Staubli VAL3: SoapTestScan.dtx

bool bSignal
bool bTxt1
bool bTxt2
bool bTxt3
bool btrig
public dio fout = {link=fOut0}
public frame FrmDraw = {x=1000, y=-50, fatherId=world[0]}
mdesc mNomSpeed
num l_nInit = 1500
public num nByteOut[48]
num nNumTotal = 5031
num nNumrecord = 5031
public num nTranC[6]
  [0] = -21.496
  [1] = -9.92
  [2] = 104.826
  [3] = 179.902
  [4] = 0.184
  [5] = -123.901
num nTxtTotal = 11
num n_sTxt = 1
num ndelay = 91.328
public num nnnn
num ntime = 653.375
public pointRx shere = {x=-21.496, y=-9.92, z=104.826, rx=179.902, ry=0.184, rz=-123.901, fatherId=FrmDraw[0]}
public sio sSocketout = {link=Socket\CServerSocket}
tool tTool = {fatherId=flange[0], ioLink=valve1}
public num hpn
public num lpn
public num ppn
num very
public num hery
public num pery
public num zmin
public num ymin
public num xmin
public num zmax
public num ymax
public num xmax
public num ztp
public num ytp
public num xtp
public num xore
public num yore
public num zore
public num nMenu
public num Qery
string sTap[3000]
string sString[1500]
public pointRx pfrmCad[1500]
  [0] = {fatherId=world[0]}
  [1] = {fatherId=world[0]}
  [2] = {fatherId=world[0]}
  [3] = {fatherId=world[0]}
  [4] = {fatherId=world[0]}
  [5] = {fatherId=world[0]}
  [6] = {fatherId=world[0]}
  [7] = {fatherId=world[0]}
  [8] = {fatherId=world[0]}
  [9] = {fatherId=world[0]}
  [10] = {fatherId=world[0]}
  [11] = {fatherId=world[0]}
  [12] = {fatherId=world[0]}
  [13] = {fatherId=world[0]}
  [14] = {fatherId=world[0]}
  [15] = {fatherId=world[0]}
  [16] = {fatherId=world[0]}
  [17] = {fatherId=world[0]}
  [18] = {fatherId=world[0]}
  [19] = {fatherId=world[0]}
  [20] = {fatherId=world[0]}
  [21] = {fatherId=world[0]}
  [22] = {fatherId=world[0]}
  [23] = {fatherId=world[0]}
  [24] = {fatherId=world[0]}
  [25] = {fatherId=world[0]}
  [26] = {fatherId=world[0]}
  [27] = {fatherId=world[0]}
  [28] = {fatherId=world[0]}
  [29] = {fatherId=world[0]}
  [30] = {fatherId=world[0]}
  [31] = {fatherId=world[0]}
  [32] = {fatherId=world[0]}
  [33] = {fatherId=world[0]}
  [34] = {fatherId=world[0]}
  [35] = {fatherId=world[0]}
  [36] = {fatherId=world[0]}
  [37] = {fatherId=world[0]}
  [38] = {fatherId=world[0]}
  [39] = {fatherId=world[0]}
  [40] = {fatherId=world[0]}
  [41] = {fatherId=world[0]}
  [42] = {fatherId=world[0]}
  [43] = {fatherId=world[0]}
  [44] = {fatherId=world[0]}
  [45] = {fatherId=world[0]}
  [46] = {fatherId=world[0]}
  [47] = {fatherId=world[0]}
  [48] = {fatherId=world[0]}
  [49] = {fatherId=world[0]}
  [50] = {fatherId=world[0]}
  [51] = {fatherId=world[0]}
  [52] = {fatherId=world[0]}
  [53] = {fatherId=world[0]}
  [54] = {fatherId=world[0]}
  [55] = {fatherId=world[0]}
  [56] = {fatherId=world[0]}
  [57] = {fatherId=world[0]}
  [58] = {fatherId=world[0]}
  [59] = {fatherId=world[0]}
  [60] = {fatherId=world[0]}
  [61] = {fatherId=world[0]}
  [62] = {fatherId=world[0]}
  [63] = {fatherId=world[0]}
  [64] = {fatherId=world[0]}
  [65] = {fatherId=world[0]}
  [66] = {fatherId=world[0]}
  [67] = {fatherId=world[0]}
  [68] = {fatherId=world[0]}
  [69] = {fatherId=world[0]}
  [70] = {fatherId=world[0]}
  [71] = {fatherId=world[0]}
  [72] = {fatherId=world[0]}
  [73] = {fatherId=world[0]}
  [74] = {fatherId=world[0]}
  [75] = {fatherId=world[0]}
  [76] = {fatherId=world[0]}
  [77] = {fatherId=world[0]}
  [78] = {fatherId=world[0]}
  [79] = {fatherId=world[0]}
  [80] = {fatherId=world[0]}
  [81] = {fatherId=world[0]}
  [82] = {fatherId=world[0]}
  [83] = {fatherId=world[0]}
  [84] = {fatherId=world[0]}
  [85] = {fatherId=world[0]}
  [86] = {fatherId=world[0]}
  [87] = {fatherId=world[0]}
  [88] = {fatherId=world[0]}
  [89] = {fatherId=world[0]}
  [90] = {fatherId=world[0]}
  [91] = {fatherId=world[0]}
  [92] = {fatherId=world[0]}
  [93] = {fatherId=world[0]}
  [94] = {fatherId=world[0]}
  [95] = {fatherId=world[0]}
  [96] = {fatherId=world[0]}
  [97] = {fatherId=world[0]}
  [98] = {fatherId=world[0]}
  [99] = {fatherId=world[0]}
  [100] = {fatherId=world[0]}
  [101] = {fatherId=world[0]}
  [102] = {fatherId=world[0]}
  [103] = {fatherId=world[0]}
  [104] = {fatherId=world[0]}
  [105] = {fatherId=world[0]}
  [106] = {fatherId=world[0]}
  [107] = {fatherId=world[0]}
  [108] = {fatherId=world[0]}
  [109] = {fatherId=world[0]}
  [110] = {fatherId=world[0]}
  [111] = {fatherId=world[0]}
  [112] = {fatherId=world[0]}
  [113] = {fatherId=world[0]}
  [114] = {fatherId=world[0]}
  [115] = {fatherId=world[0]}
  [116] = {fatherId=world[0]}
  [117] = {fatherId=world[0]}
  [118] = {fatherId=world[0]}
  [119] = {fatherId=world[0]}
  [120] = {fatherId=world[0]}
  [121] = {fatherId=world[0]}
  [122] = {fatherId=world[0]}
  [123] = {fatherId=world[0]}
  [124] = {fatherId=world[0]}
  [125] = {fatherId=world[0]}
  [126] = {fatherId=world[0]}
  [127] = {fatherId=world[0]}
  [128] = {fatherId=world[0]}
  [129] = {fatherId=world[0]}
  [130] = {fatherId=world[0]}
  [131] = {fatherId=world[0]}
  [132] = {fatherId=world[0]}
  [133] = {fatherId=world[0]}
  [134] = {fatherId=world[0]}
  [135] = {fatherId=world[0]}
  [136] = {fatherId=world[0]}
  [137] = {fatherId=world[0]}
  [138] = {fatherId=world[0]}
  [139] = {fatherId=world[0]}
  [140] = {fatherId=world[0]}
  [141] = {fatherId=world[0]}
  [142] = {fatherId=world[0]}
  [143] = {fatherId=world[0]}
  [144] = {fatherId=world[0]}
  [145] = {fatherId=world[0]}
  [146] = {fatherId=world[0]}
  [147] = {fatherId=world[0]}
  [148] = {fatherId=world[0]}
  [149] = {fatherId=world[0]}
  [150] = {fatherId=world[0]}
  [151] = {fatherId=world[0]}
  [152] = {fatherId=world[0]}
  [153] = {fatherId=world[0]}
  [154] = {fatherId=world[0]}
  [155] = {fatherId=world[0]}
  [156] = {fatherId=world[0]}
  [157] = {fatherId=world[0]}
  [158] = {fatherId=world[0]}
  [159] = {fatherId=world[0]}
  [160] = {fatherId=world[0]}
  [161] = {fatherId=world[0]}
  [162] = {fatherId=world[0]}
  [163] = {fatherId=world[0]}
  [164] = {fatherId=world[0]}
  [165] = {fatherId=world[0]}
  [166] = {fatherId=world[0]}
  [167] = {fatherId=world[0]}
  [168] = {fatherId=world[0]}
  [169] = {fatherId=world[0]}
  [170] = {fatherId=world[0]}
  [171] = {fatherId=world[0]}
  [172] = {fatherId=world[0]}
  [173] = {fatherId=world[0]}
  [174] = {fatherId=world[0]}
  [175] = {fatherId=world[0]}
  [176] = {fatherId=world[0]}
  [177] = {fatherId=world[0]}
  [178] = {fatherId=world[0]}
  [179] = {fatherId=world[0]}
  [180] = {fatherId=world[0]}
  [181] = {fatherId=world[0]}
  [182] = {fatherId=world[0]}
  [183] = {fatherId=world[0]}
  [184] = {fatherId=world[0]}
  [185] = {fatherId=world[0]}
  [186] = {fatherId=world[0]}
  [187] = {fatherId=world[0]}
  [188] = {fatherId=world[0]}
  [189] = {fatherId=world[0]}
  [190] = {fatherId=world[0]}
  [191] = {fatherId=world[0]}
  [192] = {fatherId=world[0]}
  [193] = {fatherId=world[0]}
  [194] = {fatherId=world[0]}
  [195] = {fatherId=world[0]}
  [196] = {fatherId=world[0]}
  [197] = {fatherId=world[0]}
  [198] = {fatherId=world[0]}
  [199] = {fatherId=world[0]}
  [200] = {fatherId=world[0]}
  [201] = {fatherId=world[0]}
  [202] = {fatherId=world[0]}
  [203] = {fatherId=world[0]}
  [204] = {fatherId=world[0]}
  [205] = {fatherId=world[0]}
  [206] = {fatherId=world[0]}
  [207] = {fatherId=world[0]}
  [208] = {fatherId=world[0]}
  [209] = {fatherId=world[0]}
  [210] = {fatherId=world[0]}
  [211] = {fatherId=world[0]}
  [212] = {fatherId=world[0]}
  [213] = {fatherId=world[0]}
  [214] = {fatherId=world[0]}
  [215] = {fatherId=world[0]}
  [216] = {fatherId=world[0]}
  [217] = {fatherId=world[0]}
  [218] = {fatherId=world[0]}
  [219] = {fatherId=world[0]}
  [220] = {fatherId=world[0]}
  [221] = {fatherId=world[0]}
  [222] = {fatherId=world[0]}
  [223] = {fatherId=world[0]}
  [224] = {fatherId=world[0]}
  [225] = {fatherId=world[0]}
  [226] = {fatherId=world[0]}
  [227] = {fatherId=world[0]}
  [228] = {fatherId=world[0]}
  [229] = {fatherId=world[0]}
  [230] = {fatherId=world[0]}
  [231] = {fatherId=world[0]}
  [232] = {fatherId=world[0]}
  [233] = {fatherId=world[0]}
  [234] = {fatherId=world[0]}
  [235] = {fatherId=world[0]}
  [236] = {fatherId=world[0]}
  [237] = {fatherId=world[0]}
  [238] = {fatherId=world[0]}
  [239] = {fatherId=world[0]}
  [240] = {fatherId=world[0]}
  [241] = {fatherId=world[0]}
  [242] = {fatherId=world[0]}
  [243] = {fatherId=world[0]}
  [244] = {fatherId=world[0]}
  [245] = {fatherId=world[0]}
  [246] = {fatherId=world[0]}
  [247] = {fatherId=world[0]}
  [248] = {fatherId=world[0]}
  [249] = {fatherId=world[0]}
  [250] = {fatherId=world[0]}
  [251] = {fatherId=world[0]}
  [252] = {fatherId=world[0]}
  [253] = {fatherId=world[0]}
  [254] = {fatherId=world[0]}
  [255] = {fatherId=world[0]}
  [256] = {fatherId=world[0]}
  [257] = {fatherId=world[0]}
  [258] = {fatherId=world[0]}
  [259] = {fatherId=world[0]}
  [260] = {fatherId=world[0]}
  [261] = {fatherId=world[0]}
  [262] = {fatherId=world[0]}
  [263] = {fatherId=world[0]}
  [264] = {fatherId=world[0]}
  [265] = {fatherId=world[0]}
  [266] = {fatherId=world[0]}
  [267] = {fatherId=world[0]}
  [268] = {fatherId=world[0]}
  [269] = {fatherId=world[0]}
  [270] = {fatherId=world[0]}
  [271] = {fatherId=world[0]}
  [272] = {fatherId=world[0]}
  [273] = {fatherId=world[0]}
  [274] = {fatherId=world[0]}
  [275] = {fatherId=world[0]}
  [276] = {fatherId=world[0]}
  [277] = {fatherId=world[0]}
  [278] = {fatherId=world[0]}
  [279] = {fatherId=world[0]}
  [280] = {fatherId=world[0]}
  [281] = {fatherId=world[0]}
  [282] = {fatherId=world[0]}
  [283] = {fatherId=world[0]}
  [284] = {fatherId=world[0]}
  [285] = {fatherId=world[0]}
  [286] = {fatherId=world[0]}
  [287] = {fatherId=world[0]}
  [288] = {fatherId=world[0]}
  [289] = {fatherId=world[0]}
  [290] = {fatherId=world[0]}
  [291] = {fatherId=world[0]}
  [292] = {fatherId=world[0]}
  [293] = {fatherId=world[0]}
  [294] = {fatherId=world[0]}
  [295] = {fatherId=world[0]}
  [296] = {fatherId=world[0]}
  [297] = {fatherId=world[0]}
  [298] = {fatherId=world[0]}
  [299] = {fatherId=world[0]}
  [300] = {fatherId=world[0]}
  [301] = {fatherId=world[0]}
  [302] = {fatherId=world[0]}
  [303] = {fatherId=world[0]}
  [304] = {fatherId=world[0]}
  [305] = {fatherId=world[0]}
  [306] = {fatherId=world[0]}
  [307] = {fatherId=world[0]}
  [308] = {fatherId=world[0]}
  [309] = {fatherId=world[0]}
  [310] = {fatherId=world[0]}
  [311] = {fatherId=world[0]}
  [312] = {fatherId=world[0]}
  [313] = {fatherId=world[0]}
  [314] = {fatherId=world[0]}
  [315] = {fatherId=world[0]}
  [316] = {fatherId=world[0]}
  [317] = {fatherId=world[0]}
  [318] = {fatherId=world[0]}
  [319] = {fatherId=world[0]}
  [320] = {fatherId=world[0]}
  [321] = {fatherId=world[0]}
  [322] = {fatherId=world[0]}
  [323] = {fatherId=world[0]}
  [324] = {fatherId=world[0]}
  [325] = {fatherId=world[0]}
  [326] = {fatherId=world[0]}
  [327] = {fatherId=world[0]}
  [328] = {fatherId=world[0]}
  [329] = {fatherId=world[0]}
  [330] = {fatherId=world[0]}
  [331] = {fatherId=world[0]}
  [332] = {fatherId=world[0]}
  [333] = {fatherId=world[0]}
  [334] = {fatherId=world[0]}
  [335] = {fatherId=world[0]}
  [336] = {fatherId=world[0]}
  [337] = {fatherId=world[0]}
  [338] = {fatherId=world[0]}
  [339] = {fatherId=world[0]}
  [340] = {fatherId=world[0]}
  [341] = {fatherId=world[0]}
  [342] = {fatherId=world[0]}
  [343] = {fatherId=world[0]}
  [344] = {fatherId=world[0]}
  [345] = {fatherId=world[0]}
  [346] = {fatherId=world[0]}
  [347] = {fatherId=world[0]}
  [348] = {fatherId=world[0]}
  [349] = {fatherId=world[0]}
  [350] = {fatherId=world[0]}
  [351] = {fatherId=world[0]}
  [352] = {fatherId=world[0]}
  [353] = {fatherId=world[0]}
  [354] = {fatherId=world[0]}
  [355] = {fatherId=world[0]}
  [356] = {fatherId=world[0]}
  [357] = {fatherId=world[0]}
  [358] = {fatherId=world[0]}
  [359] = {fatherId=world[0]}
  [360] = {fatherId=world[0]}
  [361] = {fatherId=world[0]}
  [362] = {fatherId=world[0]}
  [363] = {fatherId=world[0]}
  [364] = {fatherId=world[0]}
  [365] = {fatherId=world[0]}
  [366] = {fatherId=world[0]}
  [367] = {fatherId=world[0]}
  [368] = {fatherId=world[0]}
  [369] = {fatherId=world[0]}
  [370] = {fatherId=world[0]}
  [371] = {fatherId=world[0]}
  [372] = {fatherId=world[0]}
  [373] = {fatherId=world[0]}
  [374] = {fatherId=world[0]}
  [375] = {fatherId=world[0]}
  [376] = {fatherId=world[0]}
  [377] = {fatherId=world[0]}
  [378] = {fatherId=world[0]}
  [379] = {fatherId=world[0]}
  [380] = {fatherId=world[0]}
  [381] = {fatherId=world[0]}
  [382] = {fatherId=world[0]}
  [383] = {fatherId=world[0]}
  [384] = {fatherId=world[0]}
  [385] = {fatherId=world[0]}
  [386] = {fatherId=world[0]}
  [387] = {fatherId=world[0]}
  [388] = {fatherId=world[0]}
  [389] = {fatherId=world[0]}
  [390] = {fatherId=world[0]}
  [391] = {fatherId=world[0]}
  [392] = {fatherId=world[0]}
  [393] = {fatherId=world[0]}
  [394] = {fatherId=world[0]}
  [395] = {fatherId=world[0]}
  [396] = {fatherId=world[0]}
  [397] = {fatherId=world[0]}
  [398] = {fatherId=world[0]}
  [399] = {fatherId=world[0]}
  [400] = {fatherId=world[0]}
  [401] = {fatherId=world[0]}
  [402] = {fatherId=world[0]}
  [403] = {fatherId=world[0]}
  [404] = {fatherId=world[0]}
  [405] = {fatherId=world[0]}
  [406] = {fatherId=world[0]}
  [407] = {fatherId=world[0]}
  [408] = {fatherId=world[0]}
  [409] = {fatherId=world[0]}
  [410] = {fatherId=world[0]}
  [411] = {fatherId=world[0]}
  [412] = {fatherId=world[0]}
  [413] = {fatherId=world[0]}
  [414] = {fatherId=world[0]}
  [415] = {fatherId=world[0]}
  [416] = {fatherId=world[0]}
  [417] = {fatherId=world[0]}
  [418] = {fatherId=world[0]}
  [419] = {fatherId=world[0]}
  [420] = {fatherId=world[0]}
  [421] = {fatherId=world[0]}
  [422] = {fatherId=world[0]}
  [423] = {fatherId=world[0]}
  [424] = {fatherId=world[0]}
  [425] = {fatherId=world[0]}
  [426] = {fatherId=world[0]}
  [427] = {fatherId=world[0]}
  [428] = {fatherId=world[0]}
  [429] = {fatherId=world[0]}
  [430] = {fatherId=world[0]}
  [431] = {fatherId=world[0]}
  [432] = {fatherId=world[0]}
  [433] = {fatherId=world[0]}
  [434] = {fatherId=world[0]}
  [435] = {fatherId=world[0]}
  [436] = {fatherId=world[0]}
  [437] = {fatherId=world[0]}
  [438] = {fatherId=world[0]}
  [439] = {fatherId=world[0]}
  [440] = {fatherId=world[0]}
  [441] = {fatherId=world[0]}
  [442] = {fatherId=world[0]}
  [443] = {fatherId=world[0]}
  [444] = {fatherId=world[0]}
  [445] = {fatherId=world[0]}
  [446] = {fatherId=world[0]}
  [447] = {fatherId=world[0]}
  [448] = {fatherId=world[0]}
  [449] = {fatherId=world[0]}
  [450] = {fatherId=world[0]}
  [451] = {fatherId=world[0]}
  [452] = {fatherId=world[0]}
  [453] = {fatherId=world[0]}
  [454] = {fatherId=world[0]}
  [455] = {fatherId=world[0]}
  [456] = {fatherId=world[0]}
  [457] = {fatherId=world[0]}
  [458] = {fatherId=world[0]}
  [459] = {fatherId=world[0]}
  [460] = {fatherId=world[0]}
  [461] = {fatherId=world[0]}
  [462] = {fatherId=world[0]}
  [463] = {fatherId=world[0]}
  [464] = {fatherId=world[0]}
  [465] = {fatherId=world[0]}
  [466] = {fatherId=world[0]}
  [467] = {fatherId=world[0]}
  [468] = {fatherId=world[0]}
  [469] = {fatherId=world[0]}
  [470] = {fatherId=world[0]}
  [471] = {fatherId=world[0]}
  [472] = {fatherId=world[0]}
  [473] = {fatherId=world[0]}
  [474] = {fatherId=world[0]}
  [475] = {fatherId=world[0]}
  [476] = {fatherId=world[0]}
  [477] = {fatherId=world[0]}
  [478] = {fatherId=world[0]}
  [479] = {fatherId=world[0]}
  [480] = {fatherId=world[0]}
  [481] = {fatherId=world[0]}
  [482] = {fatherId=world[0]}
  [483] = {fatherId=world[0]}
  [484] = {fatherId=world[0]}
  [485] = {fatherId=world[0]}
  [486] = {fatherId=world[0]}
  [487] = {fatherId=world[0]}
  [488] = {fatherId=world[0]}
  [489] = {fatherId=world[0]}
  [490] = {fatherId=world[0]}
  [491] = {fatherId=world[0]}
  [492] = {fatherId=world[0]}
  [493] = {fatherId=world[0]}
  [494] = {fatherId=world[0]}
  [495] = {fatherId=world[0]}
  [496] = {fatherId=world[0]}
  [497] = {fatherId=world[0]}
  [498] = {fatherId=world[0]}
  [499] = {fatherId=world[0]}
  [500] = {fatherId=world[0]}
  [501] = {fatherId=world[0]}
  [502] = {fatherId=world[0]}
  [503] = {fatherId=world[0]}
  [504] = {fatherId=world[0]}
  [505] = {fatherId=world[0]}
  [506] = {fatherId=world[0]}
  [507] = {fatherId=world[0]}
  [508] = {fatherId=world[0]}
  [509] = {fatherId=world[0]}
  [510] = {fatherId=world[0]}
  [511] = {fatherId=world[0]}
  [512] = {fatherId=world[0]}
  [513] = {fatherId=world[0]}
  [514] = {fatherId=world[0]}
  [515] = {fatherId=world[0]}
  [516] = {fatherId=world[0]}
  [517] = {fatherId=world[0]}
  [518] = {fatherId=world[0]}
  [519] = {fatherId=world[0]}
  [520] = {fatherId=world[0]}
  [521] = {fatherId=world[0]}
  [522] = {fatherId=world[0]}
  [523] = {fatherId=world[0]}
  [524] = {fatherId=world[0]}
  [525] = {fatherId=world[0]}
  [526] = {fatherId=world[0]}
  [527] = {fatherId=world[0]}
  [528] = {fatherId=world[0]}
  [529] = {fatherId=world[0]}
  [530] = {fatherId=world[0]}
  [531] = {fatherId=world[0]}
  [532] = {fatherId=world[0]}
  [533] = {fatherId=world[0]}
  [534] = {fatherId=world[0]}
  [535] = {fatherId=world[0]}
  [536] = {fatherId=world[0]}
  [537] = {fatherId=world[0]}
  [538] = {fatherId=world[0]}
  [539] = {fatherId=world[0]}
  [540] = {fatherId=world[0]}
  [541] = {fatherId=world[0]}
  [542] = {fatherId=world[0]}
  [543] = {fatherId=world[0]}
  [544] = {fatherId=world[0]}
  [545] = {fatherId=world[0]}
  [546] = {fatherId=world[0]}
  [547] = {fatherId=world[0]}
  [548] = {fatherId=world[0]}
  [549] = {fatherId=world[0]}
  [550] = {fatherId=world[0]}
  [551] = {fatherId=world[0]}
  [552] = {fatherId=world[0]}
  [553] = {fatherId=world[0]}
  [554] = {fatherId=world[0]}
  [555] = {fatherId=world[0]}
  [556] = {fatherId=world[0]}
  [557] = {fatherId=world[0]}
  [558] = {fatherId=world[0]}
  [559] = {fatherId=world[0]}
  [560] = {fatherId=world[0]}
  [561] = {fatherId=world[0]}
  [562] = {fatherId=world[0]}
  [563] = {fatherId=world[0]}
  [564] = {fatherId=world[0]}
  [565] = {fatherId=world[0]}
  [566] = {fatherId=world[0]}
  [567] = {fatherId=world[0]}
  [568] = {fatherId=world[0]}
  [569] = {fatherId=world[0]}
  [570] = {fatherId=world[0]}
  [571] = {fatherId=world[0]}
  [572] = {fatherId=world[0]}
  [573] = {fatherId=world[0]}
  [574] = {fatherId=world[0]}
  [575] = {fatherId=world[0]}
  [576] = {fatherId=world[0]}
  [577] = {fatherId=world[0]}
  [578] = {fatherId=world[0]}
  [579] = {fatherId=world[0]}
  [580] = {fatherId=world[0]}
  [581] = {fatherId=world[0]}
  [582] = {fatherId=world[0]}
  [583] = {fatherId=world[0]}
  [584] = {fatherId=world[0]}
  [585] = {fatherId=world[0]}
  [586] = {fatherId=world[0]}
  [587] = {fatherId=world[0]}
  [588] = {fatherId=world[0]}
  [589] = {fatherId=world[0]}
  [590] = {fatherId=world[0]}
  [591] = {fatherId=world[0]}
  [592] = {fatherId=world[0]}
  [593] = {fatherId=world[0]}
  [594] = {fatherId=world[0]}
  [595] = {fatherId=world[0]}
  [596] = {fatherId=world[0]}
  [597] = {fatherId=world[0]}
  [598] = {fatherId=world[0]}
  [599] = {fatherId=world[0]}
  [600] = {fatherId=world[0]}
  [601] = {fatherId=world[0]}
  [602] = {fatherId=world[0]}
  [603] = {fatherId=world[0]}
  [604] = {fatherId=world[0]}
  [605] = {fatherId=world[0]}
  [606] = {fatherId=world[0]}
  [607] = {fatherId=world[0]}
  [608] = {fatherId=world[0]}
  [609] = {fatherId=world[0]}
  [610] = {fatherId=world[0]}
  [611] = {fatherId=world[0]}
  [612] = {fatherId=world[0]}
  [613] = {fatherId=world[0]}
  [614] = {fatherId=world[0]}
  [615] = {fatherId=world[0]}
  [616] = {fatherId=world[0]}
  [617] = {fatherId=world[0]}
  [618] = {fatherId=world[0]}
  [619] = {fatherId=world[0]}
  [620] = {fatherId=world[0]}
  [621] = {fatherId=world[0]}
  [622] = {fatherId=world[0]}
  [623] = {fatherId=world[0]}
  [624] = {fatherId=world[0]}
  [625] = {fatherId=world[0]}
  [626] = {fatherId=world[0]}
  [627] = {fatherId=world[0]}
  [628] = {fatherId=world[0]}
  [629] = {fatherId=world[0]}
  [630] = {fatherId=world[0]}
  [631] = {fatherId=world[0]}
  [632] = {fatherId=world[0]}
  [633] = {fatherId=world[0]}
  [634] = {fatherId=world[0]}
  [635] = {fatherId=world[0]}
  [636] = {fatherId=world[0]}
  [637] = {fatherId=world[0]}
  [638] = {fatherId=world[0]}
  [639] = {fatherId=world[0]}
  [640] = {fatherId=world[0]}
  [641] = {fatherId=world[0]}
  [642] = {fatherId=world[0]}
  [643] = {fatherId=world[0]}
  [644] = {fatherId=world[0]}
  [645] = {fatherId=world[0]}
  [646] = {fatherId=world[0]}
  [647] = {fatherId=world[0]}
  [648] = {fatherId=world[0]}
  [649] = {fatherId=world[0]}
  [650] = {fatherId=world[0]}
  [651] = {fatherId=world[0]}
  [652] = {fatherId=world[0]}
  [653] = {fatherId=world[0]}
  [654] = {fatherId=world[0]}
  [655] = {fatherId=world[0]}
  [656] = {fatherId=world[0]}
  [657] = {fatherId=world[0]}
  [658] = {fatherId=world[0]}
  [659] = {fatherId=world[0]}
  [660] = {fatherId=world[0]}
  [661] = {fatherId=world[0]}
  [662] = {fatherId=world[0]}
  [663] = {fatherId=world[0]}
  [664] = {fatherId=world[0]}
  [665] = {fatherId=world[0]}
  [666] = {fatherId=world[0]}
  [667] = {fatherId=world[0]}
  [668] = {fatherId=world[0]}
  [669] = {fatherId=world[0]}
  [670] = {fatherId=world[0]}
  [671] = {fatherId=world[0]}
  [672] = {fatherId=world[0]}
  [673] = {fatherId=world[0]}
  [674] = {fatherId=world[0]}
  [675] = {fatherId=world[0]}
  [676] = {fatherId=world[0]}
  [677] = {fatherId=world[0]}
  [678] = {fatherId=world[0]}
  [679] = {fatherId=world[0]}
  [680] = {fatherId=world[0]}
  [681] = {fatherId=world[0]}
  [682] = {fatherId=world[0]}
  [683] = {fatherId=world[0]}
  [684] = {fatherId=world[0]}
  [685] = {fatherId=world[0]}
  [686] = {fatherId=world[0]}
  [687] = {fatherId=world[0]}
  [688] = {fatherId=world[0]}
  [689] = {fatherId=world[0]}
  [690] = {fatherId=world[0]}
  [691] = {fatherId=world[0]}
  [692] = {fatherId=world[0]}
  [693] = {fatherId=world[0]}
  [694] = {fatherId=world[0]}
  [695] = {fatherId=world[0]}
  [696] = {fatherId=world[0]}
  [697] = {fatherId=world[0]}
  [698] = {fatherId=world[0]}
  [699] = {fatherId=world[0]}
  [700] = {fatherId=world[0]}
  [701] = {fatherId=world[0]}
  [702] = {fatherId=world[0]}
  [703] = {fatherId=world[0]}
  [704] = {fatherId=world[0]}
  [705] = {fatherId=world[0]}
  [706] = {fatherId=world[0]}
  [707] = {fatherId=world[0]}
  [708] = {fatherId=world[0]}
  [709] = {fatherId=world[0]}
  [710] = {fatherId=world[0]}
  [711] = {fatherId=world[0]}
  [712] = {fatherId=world[0]}
  [713] = {fatherId=world[0]}
  [714] = {fatherId=world[0]}
  [715] = {fatherId=world[0]}
  [716] = {fatherId=world[0]}
  [717] = {fatherId=world[0]}
  [718] = {fatherId=world[0]}
  [719] = {fatherId=world[0]}
  [720] = {fatherId=world[0]}
  [721] = {fatherId=world[0]}
  [722] = {fatherId=world[0]}
  [723] = {fatherId=world[0]}
  [724] = {fatherId=world[0]}
  [725] = {fatherId=world[0]}
  [726] = {fatherId=world[0]}
  [727] = {fatherId=world[0]}
  [728] = {fatherId=world[0]}
  [729] = {fatherId=world[0]}
  [730] = {fatherId=world[0]}
  [731] = {fatherId=world[0]}
  [732] = {fatherId=world[0]}
  [733] = {fatherId=world[0]}
  [734] = {fatherId=world[0]}
  [735] = {fatherId=world[0]}
  [736] = {fatherId=world[0]}
  [737] = {fatherId=world[0]}
  [738] = {fatherId=world[0]}
  [739] = {fatherId=world[0]}
  [740] = {fatherId=world[0]}
  [741] = {fatherId=world[0]}
  [742] = {fatherId=world[0]}
  [743] = {fatherId=world[0]}
  [744] = {fatherId=world[0]}
  [745] = {fatherId=world[0]}
  [746] = {fatherId=world[0]}
  [747] = {fatherId=world[0]}
  [748] = {fatherId=world[0]}
  [749] = {fatherId=world[0]}
  [750] = {fatherId=world[0]}
  [751] = {fatherId=world[0]}
  [752] = {fatherId=world[0]}
  [753] = {fatherId=world[0]}
  [754] = {fatherId=world[0]}
  [755] = {fatherId=world[0]}
  [756] = {fatherId=world[0]}
  [757] = {fatherId=world[0]}
  [758] = {fatherId=world[0]}
  [759] = {fatherId=world[0]}
  [760] = {fatherId=world[0]}
  [761] = {fatherId=world[0]}
  [762] = {fatherId=world[0]}
  [763] = {fatherId=world[0]}
  [764] = {fatherId=world[0]}
  [765] = {fatherId=world[0]}
  [766] = {fatherId=world[0]}
  [767] = {fatherId=world[0]}
  [768] = {fatherId=world[0]}
  [769] = {fatherId=world[0]}
  [770] = {fatherId=world[0]}
  [771] = {fatherId=world[0]}
  [772] = {fatherId=world[0]}
  [773] = {fatherId=world[0]}
  [774] = {fatherId=world[0]}
  [775] = {fatherId=world[0]}
  [776] = {fatherId=world[0]}
  [777] = {fatherId=world[0]}
  [778] = {fatherId=world[0]}
  [779] = {fatherId=world[0]}
  [780] = {fatherId=world[0]}
  [781] = {fatherId=world[0]}
  [782] = {fatherId=world[0]}
  [783] = {fatherId=world[0]}
  [784] = {fatherId=world[0]}
  [785] = {fatherId=world[0]}
  [786] = {fatherId=world[0]}
  [787] = {fatherId=world[0]}
  [788] = {fatherId=world[0]}
  [789] = {fatherId=world[0]}
  [790] = {fatherId=world[0]}
  [791] = {fatherId=world[0]}
  [792] = {fatherId=world[0]}
  [793] = {fatherId=world[0]}
  [794] = {fatherId=world[0]}
  [795] = {fatherId=world[0]}
  [796] = {fatherId=world[0]}
  [797] = {fatherId=world[0]}
  [798] = {fatherId=world[0]}
  [799] = {fatherId=world[0]}
  [800] = {fatherId=world[0]}
  [801] = {fatherId=world[0]}
  [802] = {fatherId=world[0]}
  [803] = {fatherId=world[0]}
  [804] = {fatherId=world[0]}
  [805] = {fatherId=world[0]}
  [806] = {fatherId=world[0]}
  [807] = {fatherId=world[0]}
  [808] = {fatherId=world[0]}
  [809] = {fatherId=world[0]}
  [810] = {fatherId=world[0]}
  [811] = {fatherId=world[0]}
  [812] = {fatherId=world[0]}
  [813] = {fatherId=world[0]}
  [814] = {fatherId=world[0]}
  [815] = {fatherId=world[0]}
  [816] = {fatherId=world[0]}
  [817] = {fatherId=world[0]}
  [818] = {fatherId=world[0]}
  [819] = {fatherId=world[0]}
  [820] = {fatherId=world[0]}
  [821] = {fatherId=world[0]}
  [822] = {fatherId=world[0]}
  [823] = {fatherId=world[0]}
  [824] = {fatherId=world[0]}
  [825] = {fatherId=world[0]}
  [826] = {fatherId=world[0]}
  [827] = {fatherId=world[0]}
  [828] = {fatherId=world[0]}
  [829] = {fatherId=world[0]}
  [830] = {fatherId=world[0]}
  [831] = {fatherId=world[0]}
  [832] = {fatherId=world[0]}
  [833] = {fatherId=world[0]}
  [834] = {fatherId=world[0]}
  [835] = {fatherId=world[0]}
  [836] = {fatherId=world[0]}
  [837] = {fatherId=world[0]}
  [838] = {fatherId=world[0]}
  [839] = {fatherId=world[0]}
  [840] = {fatherId=world[0]}
  [841] = {fatherId=world[0]}
  [842] = {fatherId=world[0]}
  [843] = {fatherId=world[0]}
  [844] = {fatherId=world[0]}
  [845] = {fatherId=world[0]}
  [846] = {fatherId=world[0]}
  [847] = {fatherId=world[0]}
  [848] = {fatherId=world[0]}
  [849] = {fatherId=world[0]}
  [850] = {fatherId=world[0]}
  [851] = {fatherId=world[0]}
  [852] = {fatherId=world[0]}
  [853] = {fatherId=world[0]}
  [854] = {fatherId=world[0]}
  [855] = {fatherId=world[0]}
  [856] = {fatherId=world[0]}
  [857] = {fatherId=world[0]}
  [858] = {fatherId=world[0]}
  [859] = {fatherId=world[0]}
  [860] = {fatherId=world[0]}
  [861] = {fatherId=world[0]}
  [862] = {fatherId=world[0]}
  [863] = {fatherId=world[0]}
  [864] = {fatherId=world[0]}
  [865] = {fatherId=world[0]}
  [866] = {fatherId=world[0]}
  [867] = {fatherId=world[0]}
  [868] = {fatherId=world[0]}
  [869] = {fatherId=world[0]}
  [870] = {fatherId=world[0]}
  [871] = {fatherId=world[0]}
  [872] = {fatherId=world[0]}
  [873] = {fatherId=world[0]}
  [874] = {fatherId=world[0]}
  [875] = {fatherId=world[0]}
  [876] = {fatherId=world[0]}
  [877] = {fatherId=world[0]}
  [878] = {fatherId=world[0]}
  [879] = {fatherId=world[0]}
  [880] = {fatherId=world[0]}
  [881] = {fatherId=world[0]}
  [882] = {fatherId=world[0]}
  [883] = {fatherId=world[0]}
  [884] = {fatherId=world[0]}
  [885] = {fatherId=world[0]}
  [886] = {fatherId=world[0]}
  [887] = {fatherId=world[0]}
  [888] = {fatherId=world[0]}
  [889] = {fatherId=world[0]}
  [890] = {fatherId=world[0]}
  [891] = {fatherId=world[0]}
  [892] = {fatherId=world[0]}
  [893] = {fatherId=world[0]}
  [894] = {fatherId=world[0]}
  [895] = {fatherId=world[0]}
  [896] = {fatherId=world[0]}
  [897] = {fatherId=world[0]}
  [898] = {fatherId=world[0]}
  [899] = {fatherId=world[0]}
  [900] = {fatherId=world[0]}
  [901] = {fatherId=world[0]}
  [902] = {fatherId=world[0]}
  [903] = {fatherId=world[0]}
  [904] = {fatherId=world[0]}
  [905] = {fatherId=world[0]}
  [906] = {fatherId=world[0]}
  [907] = {fatherId=world[0]}
  [908] = {fatherId=world[0]}
  [909] = {fatherId=world[0]}
  [910] = {fatherId=world[0]}
  [911] = {fatherId=world[0]}
  [912] = {fatherId=world[0]}
  [913] = {fatherId=world[0]}
  [914] = {fatherId=world[0]}
  [915] = {fatherId=world[0]}
  [916] = {fatherId=world[0]}
  [917] = {fatherId=world[0]}
  [918] = {fatherId=world[0]}
  [919] = {fatherId=world[0]}
  [920] = {fatherId=world[0]}
  [921] = {fatherId=world[0]}
  [922] = {fatherId=world[0]}
  [923] = {fatherId=world[0]}
  [924] = {fatherId=world[0]}
  [925] = {fatherId=world[0]}
  [926] = {fatherId=world[0]}
  [927] = {fatherId=world[0]}
  [928] = {fatherId=world[0]}
  [929] = {fatherId=world[0]}
  [930] = {fatherId=world[0]}
  [931] = {fatherId=world[0]}
  [932] = {fatherId=world[0]}
  [933] = {fatherId=world[0]}
  [934] = {fatherId=world[0]}
  [935] = {fatherId=world[0]}
  [936] = {fatherId=world[0]}
  [937] = {fatherId=world[0]}
  [938] = {fatherId=world[0]}
  [939] = {fatherId=world[0]}
  [940] = {fatherId=world[0]}
  [941] = {fatherId=world[0]}
  [942] = {fatherId=world[0]}
  [943] = {fatherId=world[0]}
  [944] = {fatherId=world[0]}
  [945] = {fatherId=world[0]}
  [946] = {fatherId=world[0]}
  [947] = {fatherId=world[0]}
  [948] = {fatherId=world[0]}
  [949] = {fatherId=world[0]}
  [950] = {fatherId=world[0]}
  [951] = {fatherId=world[0]}
  [952] = {fatherId=world[0]}
  [953] = {fatherId=world[0]}
  [954] = {fatherId=world[0]}
  [955] = {fatherId=world[0]}
  [956] = {fatherId=world[0]}
  [957] = {fatherId=world[0]}
  [958] = {fatherId=world[0]}
  [959] = {fatherId=world[0]}
  [960] = {fatherId=world[0]}
  [961] = {fatherId=world[0]}
  [962] = {fatherId=world[0]}
  [963] = {fatherId=world[0]}
  [964] = {fatherId=world[0]}
  [965] = {fatherId=world[0]}
  [966] = {fatherId=world[0]}
  [967] = {fatherId=world[0]}
  [968] = {fatherId=world[0]}
  [969] = {fatherId=world[0]}
  [970] = {fatherId=world[0]}
  [971] = {fatherId=world[0]}
  [972] = {fatherId=world[0]}
  [973] = {fatherId=world[0]}
  [974] = {fatherId=world[0]}
  [975] = {fatherId=world[0]}
  [976] = {fatherId=world[0]}
  [977] = {fatherId=world[0]}
  [978] = {fatherId=world[0]}
  [979] = {fatherId=world[0]}
  [980] = {fatherId=world[0]}
  [981] = {fatherId=world[0]}
  [982] = {fatherId=world[0]}
  [983] = {fatherId=world[0]}
  [984] = {fatherId=world[0]}
  [985] = {fatherId=world[0]}
  [986] = {fatherId=world[0]}
  [987] = {fatherId=world[0]}
  [988] = {fatherId=world[0]}
  [989] = {fatherId=world[0]}
  [990] = {fatherId=world[0]}
  [991] = {fatherId=world[0]}
  [992] = {fatherId=world[0]}
  [993] = {fatherId=world[0]}
  [994] = {fatherId=world[0]}
  [995] = {fatherId=world[0]}
  [996] = {fatherId=world[0]}
  [997] = {fatherId=world[0]}
  [998] = {fatherId=world[0]}
  [999] = {fatherId=world[0]}
  [1000] = {fatherId=world[0]}
  [1001] = {fatherId=world[0]}
  [1002] = {fatherId=world[0]}
  [1003] = {fatherId=world[0]}
  [1004] = {fatherId=world[0]}
  [1005] = {fatherId=world[0]}
  [1006] = {fatherId=world[0]}
  [1007] = {fatherId=world[0]}
  [1008] = {fatherId=world[0]}
  [1009] = {fatherId=world[0]}
  [1010] = {fatherId=world[0]}
  [1011] = {fatherId=world[0]}
  [1012] = {fatherId=world[0]}
  [1013] = {fatherId=world[0]}
  [1014] = {fatherId=world[0]}
  [1015] = {fatherId=world[0]}
  [1016] = {fatherId=world[0]}
  [1017] = {fatherId=world[0]}
  [1018] = {fatherId=world[0]}
  [1019] = {fatherId=world[0]}
  [1020] = {fatherId=world[0]}
  [1021] = {fatherId=world[0]}
  [1022] = {fatherId=world[0]}
  [1023] = {fatherId=world[0]}
  [1024] = {fatherId=world[0]}
  [1025] = {fatherId=world[0]}
  [1026] = {fatherId=world[0]}
  [1027] = {fatherId=world[0]}
  [1028] = {fatherId=world[0]}
  [1029] = {fatherId=world[0]}
  [1030] = {fatherId=world[0]}
  [1031] = {fatherId=world[0]}
  [1032] = {fatherId=world[0]}
  [1033] = {fatherId=world[0]}
  [1034] = {fatherId=world[0]}
  [1035] = {fatherId=world[0]}
  [1036] = {fatherId=world[0]}
  [1037] = {fatherId=world[0]}
  [1038] = {fatherId=world[0]}
  [1039] = {fatherId=world[0]}
  [1040] = {fatherId=world[0]}
  [1041] = {fatherId=world[0]}
  [1042] = {fatherId=world[0]}
  [1043] = {fatherId=world[0]}
  [1044] = {fatherId=world[0]}
  [1045] = {fatherId=world[0]}
  [1046] = {fatherId=world[0]}
  [1047] = {fatherId=world[0]}
  [1048] = {fatherId=world[0]}
  [1049] = {fatherId=world[0]}
  [1050] = {fatherId=world[0]}
  [1051] = {fatherId=world[0]}
  [1052] = {fatherId=world[0]}
  [1053] = {fatherId=world[0]}
  [1054] = {fatherId=world[0]}
  [1055] = {fatherId=world[0]}
  [1056] = {fatherId=world[0]}
  [1057] = {fatherId=world[0]}
  [1058] = {fatherId=world[0]}
  [1059] = {fatherId=world[0]}
  [1060] = {fatherId=world[0]}
  [1061] = {fatherId=world[0]}
  [1062] = {fatherId=world[0]}
  [1063] = {fatherId=world[0]}
  [1064] = {fatherId=world[0]}
  [1065] = {fatherId=world[0]}
  [1066] = {fatherId=world[0]}
  [1067] = {fatherId=world[0]}
  [1068] = {fatherId=world[0]}
  [1069] = {fatherId=world[0]}
  [1070] = {fatherId=world[0]}
  [1071] = {fatherId=world[0]}
  [1072] = {fatherId=world[0]}
  [1073] = {fatherId=world[0]}
  [1074] = {fatherId=world[0]}
  [1075] = {fatherId=world[0]}
  [1076] = {fatherId=world[0]}
  [1077] = {fatherId=world[0]}
  [1078] = {fatherId=world[0]}
  [1079] = {fatherId=world[0]}
  [1080] = {fatherId=world[0]}
  [1081] = {fatherId=world[0]}
  [1082] = {fatherId=world[0]}
  [1083] = {fatherId=world[0]}
  [1084] = {fatherId=world[0]}
  [1085] = {fatherId=world[0]}
  [1086] = {fatherId=world[0]}
  [1087] = {fatherId=world[0]}
  [1088] = {fatherId=world[0]}
  [1089] = {fatherId=world[0]}
  [1090] = {fatherId=world[0]}
  [1091] = {fatherId=world[0]}
  [1092] = {fatherId=world[0]}
  [1093] = {fatherId=world[0]}
  [1094] = {fatherId=world[0]}
  [1095] = {fatherId=world[0]}
  [1096] = {fatherId=world[0]}
  [1097] = {fatherId=world[0]}
  [1098] = {fatherId=world[0]}
  [1099] = {fatherId=world[0]}
  [1100] = {fatherId=world[0]}
  [1101] = {fatherId=world[0]}
  [1102] = {fatherId=world[0]}
  [1103] = {fatherId=world[0]}
  [1104] = {fatherId=world[0]}
  [1105] = {fatherId=world[0]}
  [1106] = {fatherId=world[0]}
  [1107] = {fatherId=world[0]}
  [1108] = {fatherId=world[0]}
  [1109] = {fatherId=world[0]}
  [1110] = {fatherId=world[0]}
  [1111] = {fatherId=world[0]}
  [1112] = {fatherId=world[0]}
  [1113] = {fatherId=world[0]}
  [1114] = {fatherId=world[0]}
  [1115] = {fatherId=world[0]}
  [1116] = {fatherId=world[0]}
  [1117] = {fatherId=world[0]}
  [1118] = {fatherId=world[0]}
  [1119] = {fatherId=world[0]}
  [1120] = {fatherId=world[0]}
  [1121] = {fatherId=world[0]}
  [1122] = {fatherId=world[0]}
  [1123] = {fatherId=world[0]}
  [1124] = {fatherId=world[0]}
  [1125] = {fatherId=world[0]}
  [1126] = {fatherId=world[0]}
  [1127] = {fatherId=world[0]}
  [1128] = {fatherId=world[0]}
  [1129] = {fatherId=world[0]}
  [1130] = {fatherId=world[0]}
  [1131] = {fatherId=world[0]}
  [1132] = {fatherId=world[0]}
  [1133] = {fatherId=world[0]}
  [1134] = {fatherId=world[0]}
  [1135] = {fatherId=world[0]}
  [1136] = {fatherId=world[0]}
  [1137] = {fatherId=world[0]}
  [1138] = {fatherId=world[0]}
  [1139] = {fatherId=world[0]}
  [1140] = {fatherId=world[0]}
  [1141] = {fatherId=world[0]}
  [1142] = {fatherId=world[0]}
  [1143] = {fatherId=world[0]}
  [1144] = {fatherId=world[0]}
  [1145] = {fatherId=world[0]}
  [1146] = {fatherId=world[0]}
  [1147] = {fatherId=world[0]}
  [1148] = {fatherId=world[0]}
  [1149] = {fatherId=world[0]}
  [1150] = {fatherId=world[0]}
  [1151] = {fatherId=world[0]}
  [1152] = {fatherId=world[0]}
  [1153] = {fatherId=world[0]}
  [1154] = {fatherId=world[0]}
  [1155] = {fatherId=world[0]}
  [1156] = {fatherId=world[0]}
  [1157] = {fatherId=world[0]}
  [1158] = {fatherId=world[0]}
  [1159] = {fatherId=world[0]}
  [1160] = {fatherId=world[0]}
  [1161] = {fatherId=world[0]}
  [1162] = {fatherId=world[0]}
  [1163] = {fatherId=world[0]}
  [1164] = {fatherId=world[0]}
  [1165] = {fatherId=world[0]}
  [1166] = {fatherId=world[0]}
  [1167] = {fatherId=world[0]}
  [1168] = {fatherId=world[0]}
  [1169] = {fatherId=world[0]}
  [1170] = {fatherId=world[0]}
  [1171] = {fatherId=world[0]}
  [1172] = {fatherId=world[0]}
  [1173] = {fatherId=world[0]}
  [1174] = {fatherId=world[0]}
  [1175] = {fatherId=world[0]}
  [1176] = {fatherId=world[0]}
  [1177] = {fatherId=world[0]}
  [1178] = {fatherId=world[0]}
  [1179] = {fatherId=world[0]}
  [1180] = {fatherId=world[0]}
  [1181] = {fatherId=world[0]}
  [1182] = {fatherId=world[0]}
  [1183] = {fatherId=world[0]}
  [1184] = {fatherId=world[0]}
  [1185] = {fatherId=world[0]}
  [1186] = {fatherId=world[0]}
  [1187] = {fatherId=world[0]}
  [1188] = {fatherId=world[0]}
  [1189] = {fatherId=world[0]}
  [1190] = {fatherId=world[0]}
  [1191] = {fatherId=world[0]}
  [1192] = {fatherId=world[0]}
  [1193] = {fatherId=world[0]}
  [1194] = {fatherId=world[0]}
  [1195] = {fatherId=world[0]}
  [1196] = {fatherId=world[0]}
  [1197] = {fatherId=world[0]}
  [1198] = {fatherId=world[0]}
  [1199] = {fatherId=world[0]}
  [1200] = {fatherId=world[0]}
  [1201] = {fatherId=world[0]}
  [1202] = {fatherId=world[0]}
  [1203] = {fatherId=world[0]}
  [1204] = {fatherId=world[0]}
  [1205] = {fatherId=world[0]}
  [1206] = {fatherId=world[0]}
  [1207] = {fatherId=world[0]}
  [1208] = {fatherId=world[0]}
  [1209] = {fatherId=world[0]}
  [1210] = {fatherId=world[0]}
  [1211] = {fatherId=world[0]}
  [1212] = {fatherId=world[0]}
  [1213] = {fatherId=world[0]}
  [1214] = {fatherId=world[0]}
  [1215] = {fatherId=world[0]}
  [1216] = {fatherId=world[0]}
  [1217] = {fatherId=world[0]}
  [1218] = {fatherId=world[0]}
  [1219] = {fatherId=world[0]}
  [1220] = {fatherId=world[0]}
  [1221] = {fatherId=world[0]}
  [1222] = {fatherId=world[0]}
  [1223] = {fatherId=world[0]}
  [1224] = {fatherId=world[0]}
  [1225] = {fatherId=world[0]}
  [1226] = {fatherId=world[0]}
  [1227] = {fatherId=world[0]}
  [1228] = {fatherId=world[0]}
  [1229] = {fatherId=world[0]}
  [1230] = {fatherId=world[0]}
  [1231] = {fatherId=world[0]}
  [1232] = {fatherId=world[0]}
  [1233] = {fatherId=world[0]}
  [1234] = {fatherId=world[0]}
  [1235] = {fatherId=world[0]}
  [1236] = {fatherId=world[0]}
  [1237] = {fatherId=world[0]}
  [1238] = {fatherId=world[0]}
  [1239] = {fatherId=world[0]}
  [1240] = {fatherId=world[0]}
  [1241] = {fatherId=world[0]}
  [1242] = {fatherId=world[0]}
  [1243] = {fatherId=world[0]}
  [1244] = {fatherId=world[0]}
  [1245] = {fatherId=world[0]}
  [1246] = {fatherId=world[0]}
  [1247] = {fatherId=world[0]}
  [1248] = {fatherId=world[0]}
  [1249] = {fatherId=world[0]}
  [1250] = {fatherId=world[0]}
  [1251] = {fatherId=world[0]}
  [1252] = {fatherId=world[0]}
  [1253] = {fatherId=world[0]}
  [1254] = {fatherId=world[0]}
  [1255] = {fatherId=world[0]}
  [1256] = {fatherId=world[0]}
  [1257] = {fatherId=world[0]}
  [1258] = {fatherId=world[0]}
  [1259] = {fatherId=world[0]}
  [1260] = {fatherId=world[0]}
  [1261] = {fatherId=world[0]}
  [1262] = {fatherId=world[0]}
  [1263] = {fatherId=world[0]}
  [1264] = {fatherId=world[0]}
  [1265] = {fatherId=world[0]}
  [1266] = {fatherId=world[0]}
  [1267] = {fatherId=world[0]}
  [1268] = {fatherId=world[0]}
  [1269] = {fatherId=world[0]}
  [1270] = {fatherId=world[0]}
  [1271] = {fatherId=world[0]}
  [1272] = {fatherId=world[0]}
  [1273] = {fatherId=world[0]}
  [1274] = {fatherId=world[0]}
  [1275] = {fatherId=world[0]}
  [1276] = {fatherId=world[0]}
  [1277] = {fatherId=world[0]}
  [1278] = {fatherId=world[0]}
  [1279] = {fatherId=world[0]}
  [1280] = {fatherId=world[0]}
  [1281] = {fatherId=world[0]}
  [1282] = {fatherId=world[0]}
  [1283] = {fatherId=world[0]}
  [1284] = {fatherId=world[0]}
  [1285] = {fatherId=world[0]}
  [1286] = {fatherId=world[0]}
  [1287] = {fatherId=world[0]}
  [1288] = {fatherId=world[0]}
  [1289] = {fatherId=world[0]}
  [1290] = {fatherId=world[0]}
  [1291] = {fatherId=world[0]}
  [1292] = {fatherId=world[0]}
  [1293] = {fatherId=world[0]}
  [1294] = {fatherId=world[0]}
  [1295] = {fatherId=world[0]}
  [1296] = {fatherId=world[0]}
  [1297] = {fatherId=world[0]}
  [1298] = {fatherId=world[0]}
  [1299] = {fatherId=world[0]}
  [1300] = {fatherId=world[0]}
  [1301] = {fatherId=world[0]}
  [1302] = {fatherId=world[0]}
  [1303] = {fatherId=world[0]}
  [1304] = {fatherId=world[0]}
  [1305] = {fatherId=world[0]}
  [1306] = {fatherId=world[0]}
  [1307] = {fatherId=world[0]}
  [1308] = {fatherId=world[0]}
  [1309] = {fatherId=world[0]}
  [1310] = {fatherId=world[0]}
  [1311] = {fatherId=world[0]}
  [1312] = {fatherId=world[0]}
  [1313] = {fatherId=world[0]}
  [1314] = {fatherId=world[0]}
  [1315] = {fatherId=world[0]}
  [1316] = {fatherId=world[0]}
  [1317] = {fatherId=world[0]}
  [1318] = {fatherId=world[0]}
  [1319] = {fatherId=world[0]}
  [1320] = {fatherId=world[0]}
  [1321] = {fatherId=world[0]}
  [1322] = {fatherId=world[0]}
  [1323] = {fatherId=world[0]}
  [1324] = {fatherId=world[0]}
  [1325] = {fatherId=world[0]}
  [1326] = {fatherId=world[0]}
  [1327] = {fatherId=world[0]}
  [1328] = {fatherId=world[0]}
  [1329] = {fatherId=world[0]}
  [1330] = {fatherId=world[0]}
  [1331] = {fatherId=world[0]}
  [1332] = {fatherId=world[0]}
  [1333] = {fatherId=world[0]}
  [1334] = {fatherId=world[0]}
  [1335] = {fatherId=world[0]}
  [1336] = {fatherId=world[0]}
  [1337] = {fatherId=world[0]}
  [1338] = {fatherId=world[0]}
  [1339] = {fatherId=world[0]}
  [1340] = {fatherId=world[0]}
  [1341] = {fatherId=world[0]}
  [1342] = {fatherId=world[0]}
  [1343] = {fatherId=world[0]}
  [1344] = {fatherId=world[0]}
  [1345] = {fatherId=world[0]}
  [1346] = {fatherId=world[0]}
  [1347] = {fatherId=world[0]}
  [1348] = {fatherId=world[0]}
  [1349] = {fatherId=world[0]}
  [1350] = {fatherId=world[0]}
  [1351] = {fatherId=world[0]}
  [1352] = {fatherId=world[0]}
  [1353] = {fatherId=world[0]}
  [1354] = {fatherId=world[0]}
  [1355] = {fatherId=world[0]}
  [1356] = {fatherId=world[0]}
  [1357] = {fatherId=world[0]}
  [1358] = {fatherId=world[0]}
  [1359] = {fatherId=world[0]}
  [1360] = {fatherId=world[0]}
  [1361] = {fatherId=world[0]}
  [1362] = {fatherId=world[0]}
  [1363] = {fatherId=world[0]}
  [1364] = {fatherId=world[0]}
  [1365] = {fatherId=world[0]}
  [1366] = {fatherId=world[0]}
  [1367] = {fatherId=world[0]}
  [1368] = {fatherId=world[0]}
  [1369] = {fatherId=world[0]}
  [1370] = {fatherId=world[0]}
  [1371] = {fatherId=world[0]}
  [1372] = {fatherId=world[0]}
  [1373] = {fatherId=world[0]}
  [1374] = {fatherId=world[0]}
  [1375] = {fatherId=world[0]}
  [1376] = {fatherId=world[0]}
  [1377] = {fatherId=world[0]}
  [1378] = {fatherId=world[0]}
  [1379] = {fatherId=world[0]}
  [1380] = {fatherId=world[0]}
  [1381] = {fatherId=world[0]}
  [1382] = {fatherId=world[0]}
  [1383] = {fatherId=world[0]}
  [1384] = {fatherId=world[0]}
  [1385] = {fatherId=world[0]}
  [1386] = {fatherId=world[0]}
  [1387] = {fatherId=world[0]}
  [1388] = {fatherId=world[0]}
  [1389] = {fatherId=world[0]}
  [1390] = {fatherId=world[0]}
  [1391] = {fatherId=world[0]}
  [1392] = {fatherId=world[0]}
  [1393] = {fatherId=world[0]}
  [1394] = {fatherId=world[0]}
  [1395] = {fatherId=world[0]}
  [1396] = {fatherId=world[0]}
  [1397] = {fatherId=world[0]}
  [1398] = {fatherId=world[0]}
  [1399] = {fatherId=world[0]}
  [1400] = {fatherId=world[0]}
  [1401] = {fatherId=world[0]}
  [1402] = {fatherId=world[0]}
  [1403] = {fatherId=world[0]}
  [1404] = {fatherId=world[0]}
  [1405] = {fatherId=world[0]}
  [1406] = {fatherId=world[0]}
  [1407] = {fatherId=world[0]}
  [1408] = {fatherId=world[0]}
  [1409] = {fatherId=world[0]}
  [1410] = {fatherId=world[0]}
  [1411] = {fatherId=world[0]}
  [1412] = {fatherId=world[0]}
  [1413] = {fatherId=world[0]}
  [1414] = {fatherId=world[0]}
  [1415] = {fatherId=world[0]}
  [1416] = {fatherId=world[0]}
  [1417] = {fatherId=world[0]}
  [1418] = {fatherId=world[0]}
  [1419] = {fatherId=world[0]}
  [1420] = {fatherId=world[0]}
  [1421] = {fatherId=world[0]}
  [1422] = {fatherId=world[0]}
  [1423] = {fatherId=world[0]}
  [1424] = {fatherId=world[0]}
  [1425] = {fatherId=world[0]}
  [1426] = {fatherId=world[0]}
  [1427] = {fatherId=world[0]}
  [1428] = {fatherId=world[0]}
  [1429] = {fatherId=world[0]}
  [1430] = {fatherId=world[0]}
  [1431] = {fatherId=world[0]}
  [1432] = {fatherId=world[0]}
  [1433] = {fatherId=world[0]}
  [1434] = {fatherId=world[0]}
  [1435] = {fatherId=world[0]}
  [1436] = {fatherId=world[0]}
  [1437] = {fatherId=world[0]}
  [1438] = {fatherId=world[0]}
  [1439] = {fatherId=world[0]}
  [1440] = {fatherId=world[0]}
  [1441] = {fatherId=world[0]}
  [1442] = {fatherId=world[0]}
  [1443] = {fatherId=world[0]}
  [1444] = {fatherId=world[0]}
  [1445] = {fatherId=world[0]}
  [1446] = {fatherId=world[0]}
  [1447] = {fatherId=world[0]}
  [1448] = {fatherId=world[0]}
  [1449] = {fatherId=world[0]}
  [1450] = {fatherId=world[0]}
  [1451] = {fatherId=world[0]}
  [1452] = {fatherId=world[0]}
  [1453] = {fatherId=world[0]}
  [1454] = {fatherId=world[0]}
  [1455] = {fatherId=world[0]}
  [1456] = {fatherId=world[0]}
  [1457] = {fatherId=world[0]}
  [1458] = {fatherId=world[0]}
  [1459] = {fatherId=world[0]}
  [1460] = {fatherId=world[0]}
  [1461] = {fatherId=world[0]}
  [1462] = {fatherId=world[0]}
  [1463] = {fatherId=world[0]}
  [1464] = {fatherId=world[0]}
  [1465] = {fatherId=world[0]}
  [1466] = {fatherId=world[0]}
  [1467] = {fatherId=world[0]}
  [1468] = {fatherId=world[0]}
  [1469] = {fatherId=world[0]}
  [1470] = {fatherId=world[0]}
  [1471] = {fatherId=world[0]}
  [1472] = {fatherId=world[0]}
  [1473] = {fatherId=world[0]}
  [1474] = {fatherId=world[0]}
  [1475] = {fatherId=world[0]}
  [1476] = {fatherId=world[0]}
  [1477] = {fatherId=world[0]}
  [1478] = {fatherId=world[0]}
  [1479] = {fatherId=world[0]}
  [1480] = {fatherId=world[0]}
  [1481] = {fatherId=world[0]}
  [1482] = {fatherId=world[0]}
  [1483] = {fatherId=world[0]}
  [1484] = {fatherId=world[0]}
  [1485] = {fatherId=world[0]}
  [1486] = {fatherId=world[0]}
  [1487] = {fatherId=world[0]}
  [1488] = {fatherId=world[0]}
  [1489] = {fatherId=world[0]}
  [1490] = {fatherId=world[0]}
  [1491] = {fatherId=world[0]}
  [1492] = {fatherId=world[0]}
  [1493] = {fatherId=world[0]}
  [1494] = {fatherId=world[0]}
  [1495] = {fatherId=world[0]}
  [1496] = {fatherId=world[0]}
  [1497] = {fatherId=world[0]}
  [1498] = {fatherId=world[0]}
  [1499] = {fatherId=world[0]}
num nNum
string l_sString
public num n_rpt
